FUNCTION_BLOCK MotorVsBase (* Composite Function Block Type *)
  (* Standard: 61499-2 *)
  (* Version 1.0.1, 2/5/2024, ApplicationLibDevTeam, Schneider Electric, First Version *)
  PACKAGE Main;
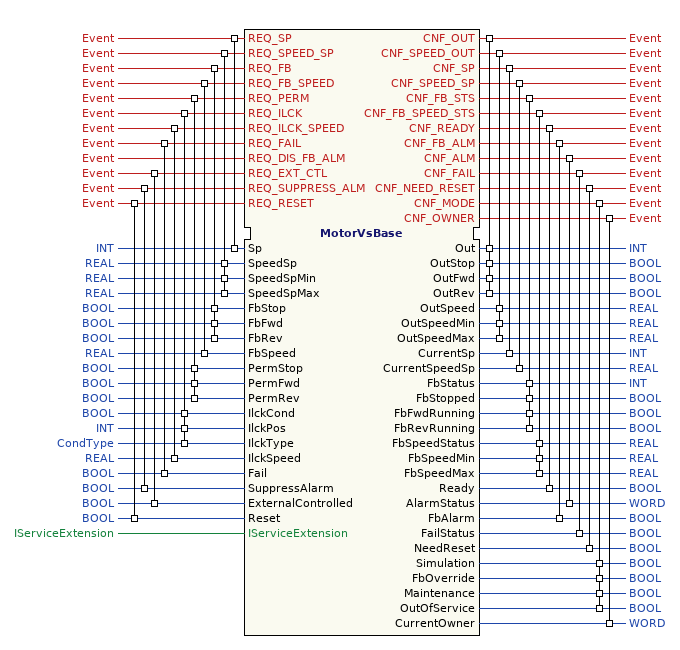
  EVENT_INPUT
    REQ_SP WITH Sp; (* Request to update setpoint *)
    REQ_SPEED_SP WITH SpeedSp, SpeedSpMin, SpeedSpMax;
    REQ_FB WITH FbStop, FbFwd, FbRev; (* Request to update feedbacks *)
    REQ_FB_SPEED WITH FbSpeed;
    REQ_PERM WITH PermStop, PermFwd, PermRev; (* Request to update permissive conditions *)
    REQ_ILCK WITH IlckCond, IlckPos, IlckType; (* Request to update interlock conditions *)
    REQ_ILCK_SPEED WITH IlckSpeed;
    REQ_FAIL WITH Fail; (* Request to update out of service and fail status and parameters *)
    REQ_DIS_FB_ALM; (* Request to disable feedback alarm *)
    REQ_EXT_CTL WITH ExternalControlled; (* Request External control signal *)
    REQ_SUPPRESS_ALM WITH SuppressAlarm; (* Request to update the alarm suppress status *)
    REQ_RESET WITH Reset; (* Request to reset the device *)
  END_EVENT
  EVENT_OUTPUT
    CNF_OUT WITH Out, OutFwd, OutStop, OutRev; (* Execution of output confirmation *)
    CNF_SPEED_OUT WITH OutSpeed, OutSpeedMin, OutSpeedMax; (* Execution of apeed output confirmation *)
    CNF_SP WITH CurrentSp; (* Execution of confirmation current setpoint *)
    CNF_SPEED_SP WITH CurrentSpeedSp; (* Execution of confirmation current speed setpoint *)
    CNF_FB_STS WITH FbFwdRunning, FbStopped, FbStatus, FbRevRunning; (* Execution of confirmed state *)
    CNF_FB_SPEED_STS WITH FbSpeedStatus, FbSpeedMin, FbSpeedMax; (* Execution of confirmed speed state *)
    CNF_READY WITH Ready; (* Execution of ready status *)
    CNF_FB_ALM WITH FbAlarm; (* Execution of confirmation  Fb alarm *)
    CNF_ALM WITH AlarmStatus; (* Execution of confirmation  alarm conditions *)
    CNF_FAIL WITH FailStatus; (* Execution of confirmation  failure *)
    CNF_NEED_RESET WITH NeedReset; (* Request for reset *)
    CNF_MODE WITH Simulation, FbOverride, Maintenance, OutOfService; (* Excecution of new operational modes *)
    CNF_OWNER WITH CurrentOwner; (* Execution confirmation of owner *)
  END_EVENT
  VAR_INPUT
    Sp : INT; (* Setpoint of device (0 = Stop, 1 = Run Forward, 2 = Run Reverse) *)
    SpeedSp : REAL; (* Speed setpoint of device *)
    SpeedSpMin : REAL; (* Speed setpoint minimum range *)
    SpeedSpMax : REAL; (* Speed setpoint maximum range *)
    FbStop : BOOL; (* 1 = Device stop feedback incoming *)
    FbFwd : BOOL; (* 1 = Device forward running feedback incoming *)
    FbRev : BOOL; (* 1 = Device reverse running feedback incoming *)
    FbSpeed : REAL; (* Device speed feedback incoming (Minimum Value  = 0.0, Maximum Value = 100.0) *)
    PermStop : BOOL := TRUE; (* 1 = Device stop permission active *)
    PermFwd : BOOL := TRUE; (* 1 = Device forward run permission active *)
    PermRev : BOOL := TRUE; (* 1 = Device reverse run permission active *)
    IlckCond : BOOL; (* 1 = Interlock condition active *)
    IlckPos : INT; (* Interlock setpoint state (0 = Stop, 1 = Run Forward, 1 = Run Reverse, 3 = Interlock inactive) *)
    IlckType : CondType; (* Type of condition interlock, (0 = Normal, 1 = Process interlock/Sequence interlock) *)
    IlckSpeed : REAL; (* Interlock speed setpoint *)
    Fail : BOOL; (* 1 = Failure is active *)
    SuppressAlarm : BOOL; (* 1 = Suppress alarm in HMI *)
    ExternalControlled : BOOL; (* 1 = External control is active *)
    Reset : BOOL; (* 1 = Reset device failure *)
  END_VAR
  VAR_OUTPUT
    Out : INT; (* Calculated output of the device ( 0 = Stop command, 1 = Forward Run command,  1 = Reverse Run command) *)
    OutStop : BOOL; (* 1 = Stop output of the device *)
    OutFwd : BOOL; (* 1 = Forward output of the device *)
    OutRev : BOOL; (* 1 = Reverse output of the device *)
    OutSpeed : REAL; (* Calculated speed output of the device *)
    OutSpeedMin : REAL; (* Current output speed minimum value *)
    OutSpeedMax : REAL; (* Current output speed maximum value *)
    CurrentSp : INT; (* Current output value considering permissive conditions *)
    CurrentSpeedSp : REAL; (* Current output value *)
    FbStatus : INT; (* Confirmed state of the device (0 = Stopped, 1 =Running, 253 = Unknown) *)
    FbStopped : BOOL; (* 1 = Stopped *)
    FbFwdRunning : BOOL; (* 1 = Running Forward *)
    FbRevRunning : BOOL; (* 1 = Running Reverse *)
    FbSpeedStatus : REAL; (* Speed feedback *)
    FbSpeedMin : REAL; (* Minimum speed setpoint range *)
    FbSpeedMax : REAL; (* Maximum speed setpoint range *)
    Ready : BOOL; (* 1 = Device is ready to run *)
    AlarmStatus : WORD; (* Bit 1 = Device failure status, Bit 2 = Feedback failure status *)
    FbAlarm : BOOL; (* Current output speed minimum value *)
    FailStatus : BOOL; (* 1 = Fail active *)
    NeedReset : BOOL; (* 1 = Device need reset to resume the operation *)
    Simulation : BOOL; (* 1 = Simulation mode is active *)
    FbOverride : BOOL; (* 1 = Feedback overide (Sp = FbStatus) *)
    Maintenance : BOOL; (* 1 = Maintenance mode is active *)
    OutOfService : BOOL; (* 1 = Out of service mode is active *)
    CurrentOwner : WORD; (* Current owner data from externlal source and basic owner 16#8 = Program owner, 16#10 = Operator owner, 16#4 = program Local and 16#40 Operator Local *)
  END_VAR
  SOCKETS
    IServiceExtension : IServiceExtension(ServiceState := TRUE); (* Services extension adapter(Seq control, Local panel, Maintenance and Owner) *)
  END_SOCKETS
  (* Alarm Managment *)
  (* Control *)
  (* Data exchange with sequence *)
  (* Initialization *)
  (* Supervision Interface *)
  (* Owner & Setpoint Management *)
  (* Speed Input *)
  (* Comment If external owner is enabled, the owner for speed selection will be decoupled from normal owner. The external speed owner can be configured from HMI *)
  FBS
    plcStart : plcStart(Delay := T#0ms, Prio := 16);
    IThis : MotorVsBase_HMI(QI := TRUE);
    spSelection : devInSel(EnBumpless2 := TRUE, EnBumpless3 := FALSE); {SET_ATTRIBUTE(Configuration.Component.HideUnusedPorts, )}
    control : motorVsLogic; {SET_ATTRIBUTE(Configuration.Component.HideUnusedPorts, )}
    basicOwner : ownerControl;
    deviceFailure : stateAlarmBasic(AlarmState := TRUE); {SET_ATTRIBUTE(HMI.AlarmText, $key:SE.App2CommonProcess.AlmLableMotorFail)}
    feedbackFailure : stateAlarmBasic(AlarmState := TRUE); {SET_ATTRIBUTE(HMI.AlarmText, $key:SE.App2CommonProcess.AlarmLabelFbFail)}
    programSpSelection : SELECT_24363B89CFDE21263; {SET_ATTRIBUTE(Configuration.GenericFBType.InterfaceParams, Runtime.Standard#CNT:=2;SELECT:BOOL;IN${CNT$}:INT)}
    speedOwner : externalOwnerSel(pin_0E0839046EC8AB65 := TRUE); {SET_ATTRIBUTE(Configuration.Component.HideUnusedPorts, )}
    speedSpSelection : devRealSel(EnBumpless2 := TRUE, EnBumpless3 := FALSE); {SET_ATTRIBUTE(Configuration.Component.HideUnusedPorts, )}
    programSpeedSpSelection : SELECT_218F0E76F8A148ECD; {SET_ATTRIBUTE(Configuration.GenericFBType.InterfaceParams, Runtime.Standard#CNT:=2;SELECT:BOOL;IN${CNT$}:REAL)}
    speedFbScale : limitScaleValue(EnScale := TRUE, UseCutoff := TRUE); {SET_ATTRIBUTE(Configuration.Component.HideUnusedPorts, )}
    speedSpRangeSel : externalRangeSel;
    resetConditions : DS_SELECTX_1579ED5B8ACDFC94C; {SET_ATTRIBUTE(Configuration.GenericFBType.InterfaceParams, Runtime.Standard#CNTX:=3;CNTY:=1;DI${CNTX,_,CNTY$}:BOOL)}
  END_FBS
  EVENT_CONNECTIONS
    spSelection.CNF TO control.REQ_SP;
    control.CNF_OUT TO IServiceExtension.CNF_STATUS;
    control.CNF_FB_STS TO IServiceExtension.CNF_STATUS;
    spSelection.CNF TO IServiceExtension.CNF_STATUS;
    control.CNF_FB_ALM TO CNF_FB_ALM;
    control.CNF_READY TO IServiceExtension.CNF_READY;
    control.CNF_MODE TO IServiceExtension.CNF_OPMODE;
    REQ_SUPPRESS_ALM TO IServiceExtension.CNF_SUPPRESS_ALM;
    REQ_SUPPRESS_ALM TO deviceFailure.REQ_SUPRESS;
    control.CNF_FB_STS TO CNF_FB_STS;
    control.CNF_OUT TO CNF_OUT;
    control.CNF_MODE TO CNF_MODE;
    REQ_FB TO control.REQ_FB;
    REQ_FAIL TO control.REQ_FAIL;
    REQ_DIS_FB_ALM TO control.REQ_PARA;
    deviceFailure.INITO TO feedbackFailure.INIT;
    REQ_PERM TO spSelection.REQ_SEL;
    IServiceExtension.REQ_OWNER TO basicOwner.REQ_STDOWNER;
    basicOwner.CNF_OWNER TO spSelection.REQ_SEL;
    feedbackFailure.INITO TO plcStart.ACK_FIRST;
    control.CNF_NEED_RESET TO CNF_NEED_RESET;
    control.CNF_READY TO CNF_READY;
    spSelection.CNF TO CNF_SP;
    REQ_EXT_CTL TO control.REQ_EXT_CTL;
    control.CNF_FAIL TO deviceFailure.REQ;
    control.CNF_FAIL TO CNF_FAIL;
    plcStart.FIRST_INIT TO IServiceExtension.CNF_SERVICE;
    control.CNF_FB_ALM TO feedbackFailure.REQ;
    control.CNF_ALM TO CNF_ALM;
    control.CNF_ILCK TO spSelection.REQ_SEL;
    control.CNF_FAIL TO spSelection.RESET_SP;
    REQ_SUPPRESS_ALM TO feedbackFailure.REQ_SUPRESS;
    REQ_PERM TO IServiceExtension.CNF_READY;
    basicOwner.CNF_OWNER TO speedOwner.REQ;
    control.CNF_FAIL TO speedSpSelection.RESET_SP;
    REQ_SPEED_SP TO programSpeedSpSelection.REQ;
    IServiceExtension.REQ_SP TO programSpeedSpSelection.REQ;
    control.CNF_ILCK TO speedSpSelection.REQ_SEL;
    speedSpSelection.CNF TO control.REQ_SPEED_SP;
    REQ_ILCK_SPEED TO speedSpSelection.REQ_SEL;
    speedOwner.CNF TO speedSpSelection.REQ_SEL;
    speedFbScale.CNF TO CNF_FB_SPEED_STS;
    IServiceExtension.REQ_OWNER TO speedOwner.REQ;
    REQ_FB_SPEED TO speedFbScale.REQ;
    speedFbScale.CNF TO IServiceExtension.CNF_PV;
    control.CNF_SPEED_OUT TO CNF_SPEED_OUT;
    speedSpSelection.CNF TO CNF_SPEED_SP;
    control.CNF_SPEED_OUT TO IServiceExtension.CNF_SP_OP;
    speedSpSelection.CNF TO IServiceExtension.CNF_SP_OP;
    programSpeedSpSelection.CNF TO speedSpSelection.REQ_SP3;
    REQ_SP TO programSpSelection.REQ;
    IServiceExtension.REQ_CMD TO programSpSelection.REQ;
    programSpSelection.CNF TO spSelection.REQ_SP3;
    control.CNF_ILCK TO IServiceExtension.CNF_READY;
    control.CNF_ALM TO IServiceExtension.CNF_READY;
    control.CNF_NEED_RESET TO IServiceExtension.CNF_READY;
    REQ_ILCK_SPEED TO control.REQ_ILCK_SPEED;
    basicOwner.CNF_OWNER TO speedSpRangeSel.REQ_SELECT;
    speedSpRangeSel.CNF TO control.REQ_SPEED_SP;
    REQ_SPEED_SP TO speedSpRangeSel.REQ_3;
    speedSpRangeSel.CNF TO speedFbScale.REQ;
    IServiceExtension.REQ_SP TO speedSpRangeSel.REQ_2;
    plcStart.FIRST_INIT TO IThis.34A017503AC1070A;
    IThis.377462E9CE5193B5 TO IThis.F2953B6BB9388F21;
    control.CNF_FB_STS TO IThis.EC791CA6E67D66B3;
    control.CNF_OUT TO IThis.EC791CA6E67D66B3;
    control.CNF_NEED_RESET TO IThis.EC791CA6E67D66B3;
    spSelection.CNF TO IThis.EC791CA6E67D66B3;
    control.CNF_TRANS_FB TO IThis.EC791CA6E67D66B3;
    REQ_SUPPRESS_ALM TO IThis.EC791CA6E67D66B3;
    deviceFailure.CNF_ALM TO IThis.EC791CA6E67D66B3;
    feedbackFailure.CNF_ALM TO IThis.EC791CA6E67D66B3;
    control.CNF_FAIL TO IThis.EC791CA6E67D66B3;
    control.CNF_ILCK TO IThis.EC791CA6E67D66B3;
    REQ_PERM TO IThis.EC791CA6E67D66B3;
    basicOwner.CNF_OWNER TO IThis.EC791CA6E67D66B3;
    speedFbScale.CNF TO IThis.EC791CA6E67D66B3;
    control.CNF_SPEED_OUT TO IThis.EC791CA6E67D66B3;
    speedOwner.CNF TO IThis.EC791CA6E67D66B3;
    speedSpSelection.CNF TO IThis.EC791CA6E67D66B3;
    speedSpRangeSel.CNF TO IThis.EC791CA6E67D66B3;
    control.PASSIVE_T TO IThis.FD2B6A321910142C;
    IThis.377462E9CE5193B5 TO deviceFailure.INIT;
    IThis.377462E9CE5193B5 TO basicOwner.REQ_BASICOWNER;
    IThis.B42FC414051FE233 TO basicOwner.REQ_BASICOWNER;
    IThis.1E115F107370F478 TO speedOwner.REQ;
    IThis.1E115F107370F478 TO IServiceExtension.CNF_OWNER;
    IThis.95BEA68906019444 TO control.REQ_PARA;
    IThis.95BEA68906019444 TO feedbackFailure.REQ_PARA;
    IThis.95BEA68906019444 TO deviceFailure.REQ_PARA;
    IThis.95BEA68906019444 TO speedSpRangeSel.REQ_SELECT;
    IThis.A8EC0BB0D1766C60 TO speedSpRangeSel.REQ_1;
    IThis.4BC263E0581D4DDB TO control.REQ_SPEED_SP;
    IThis.C6CA4032A5F6989A TO spSelection.REQ_SP2;
    IThis.369F8CFFBEE23AB4 TO speedSpSelection.REQ_SP2;
    IThis.4711DA9A2DFC024 TO basicOwner.REQ_FORCE;
    IThis.4711DA9A2DFC024 TO control.REQ_PARA;
    IThis.4711DA9A2DFC024 TO spSelection.REQ_SEL;
    IThis.4711DA9A2DFC024 TO speedSpSelection.REQ_SEL;
    REQ_ILCK TO control.REQ_ILCK;
    REQ_EXT_CTL TO IThis.EC791CA6E67D66B3;
    basicOwner.CNF_OWNER TO CNF_OWNER;
    REQ_RESET TO resetConditions.REQ3;
    IServiceExtension.REQ_RESET TO resetConditions.REQ2;
    IThis.1A2B085F4B246BF1 TO resetConditions.REQ1;
    resetConditions.IND TO control.REQ_RESET;
    IThis.95BEA68906019444 TO IServiceExtension.CNF_CFG;
    IThis.A8EC0BB0D1766C60 TO speedFbScale.REQ;
  END_CONNECTIONS
  DATA_CONNECTIONS
    spSelection.PermVal TO control.Sp;
    control.FbStatus TO IServiceExtension.Status;
    spSelection.PermVal TO IServiceExtension.CurrentSp;
    control.Out TO IServiceExtension.CurrentOp;
    control.NeedReset TO IServiceExtension.NeedReset;
    control.FbAlarm TO FbAlarm;
    control.Mode TO IServiceExtension.OpMode;
    control.Ready TO IServiceExtension.Ready;
    SuppressAlarm TO IServiceExtension.SuppressAlarm;
    SuppressAlarm TO deviceFailure.Suppress;
    SuppressAlarm TO feedbackFailure.Suppress;
    control.FbAlarm TO feedbackFailure.Input;
    control.FailStatus TO FailStatus;
    IlckPos TO control.IlckPos;
    IlckType TO control.IlckType;
    FbStop TO control.FbStop;
    FbFwd TO control.FbFwd;
    Fail TO control.Fail;
    PermStop TO spSelection.PermPassive;
    PermFwd TO spSelection.PermActive1;
    control.FbStopped TO FbStopped;
    control.FbFwdRunning TO FbFwdRunning;
    control.Out TO Out;
    control.FbStatus TO FbStatus;
    basicOwner.ProgramOwner TO spSelection.Sel3;
    basicOwner.OperatorOwner TO spSelection.Sel2;
    IlckPos TO spSelection.IlckSp;
    control.Interlocked TO spSelection.Ilck;
    IServiceExtension.StdOwner TO basicOwner.StdOwner;
    basicOwner.StdOwnerConnected TO programSpSelection.SELECT;
    control.NeedReset TO NeedReset;
    control.Ready TO Ready;
    ExternalControlled TO control.ExternalControlled;
    control.FailStatus TO deviceFailure.Input;
    control.AlarmStatus TO AlarmStatus;
    spSelection.PermVal TO CurrentSp;
    control.FailStatus TO spSelection.Fail;
    PermStop TO IServiceExtension.PermPassive;
    PermFwd TO IServiceExtension.PermActive1;
    control.AlarmStatus TO IServiceExtension.Alarm;
    control.Interlocked TO IServiceExtension.Interlocked;
    PermRev TO spSelection.PermActive2;
    basicOwner.Owner TO speedOwner.StdOwner;
    speedOwner.OperOwner TO speedSpSelection.Sel2;
    speedOwner.ProgOwner TO speedSpSelection.Sel3;
    control.Interlocked TO speedSpSelection.Ilck;
    control.FailStatus TO speedSpSelection.Fail;
    basicOwner.StdOwnerConnected TO programSpeedSpSelection.SELECT;
    control.FbRevRunning TO FbRevRunning;
    FbRev TO control.FbRev;
    speedSpSelection.CurrentVal TO control.SpeedSp;
    IlckSpeed TO control.IlckSpeed;
    IlckSpeed TO speedSpSelection.IlckSp;
    speedSpSelection.CurrentVal TO IServiceExtension.CurrentSpReal;
    speedFbScale.PvOut TO FbSpeedStatus;
    control.OutSpeed TO IServiceExtension.CurrentOpReal1;
    speedFbScale.PvOut TO IServiceExtension.Pv;
    IServiceExtension.ExtOwner TO speedOwner.ExtOwner;
    FbSpeed TO speedFbScale.PvIn;
    control.OutSpeedScaled TO OutSpeed;
    speedSpSelection.CurrentVal TO CurrentSpeedSp;
    PermRev TO IServiceExtension.PermActive2;
    SpeedSp TO programSpeedSpSelection.IN1;
    IServiceExtension.SpReal1 TO programSpeedSpSelection.IN2;
    programSpeedSpSelection.OUT TO speedSpSelection.Val3;
    Sp TO programSpSelection.IN1;
    IServiceExtension.Sp TO programSpSelection.IN2;
    programSpSelection.OUT TO spSelection.Val3;
    control.OutFwd TO OutFwd;
    control.OutStop TO OutStop;
    control.OutRev TO OutRev;
    speedSpRangeSel.RangeMin TO control.SpeedSpMin;
    speedSpRangeSel.RangeMin TO speedFbScale.CutoffValue;
    speedSpRangeSel.RangeMin TO speedFbScale.OutMin;
    speedSpRangeSel.RangeMin TO FbSpeedMin;
    speedSpRangeSel.RangeMax TO control.SpeedSpMax;
    speedSpRangeSel.RangeMax TO speedFbScale.OutMax;
    speedSpRangeSel.RangeMax TO FbSpeedMax;
    basicOwner.StdOwnerConnected TO speedSpRangeSel.StdOwnerConnected;
    IServiceExtension.RangeMin TO speedSpRangeSel.RangeMin2;
    IServiceExtension.RangeMax TO speedSpRangeSel.RangeMax2;
    SpeedSpMin TO speedSpRangeSel.RangeMin3;
    SpeedSpMax TO speedSpRangeSel.RangeMax3;
    control.FbStatus TO IThis.E35507CB164A688E;
    control.TransFbStatus TO IThis.937CA40F4D16204B;
    speedFbScale.PvOut TO IThis.5FDD97900C8D5AF7;
    spSelection.PermVal TO IThis.C6876D790F3A950E;
    control.Out TO IThis.D2C35BC47DF71FCC;
    speedSpSelection.CurrentVal TO IThis.977C6234F7727BFD;
    speedSpRangeSel.RangeMin TO IThis.51D483D786BBCC80;
    speedSpRangeSel.RangeMax TO IThis.4209B267B5CDF46;
    control.OutSpeedScaled TO IThis.53DD13BB8E7CA9FB;
    basicOwner.Owner TO IThis.9CB24E1B5B149DBC;
    speedOwner.Owner TO IThis.A2BE276F0EB32372;
    control.NeedReset TO IThis.9CD6749867E91606;
    control.Interlocked TO IThis.22A0744EA4DC0124;
    feedbackFailure.AlarmStatus TO IThis.7F794E74835A9A2;
    deviceFailure.AlarmStatus TO IThis.E4BB2C7DF94BE70A;
    PermStop TO IThis.AB1D2B96094C90BD;
    PermFwd TO IThis.18DA785EF50AD374;
    PermRev TO IThis.49F3F7DCC2A083AE;
    control.PassiveRemainTime TO IThis.1956BBB3F5CBD486;
    basicOwner.StdOwnerConnected TO IThis.621B2EAA60B4DCF6;
    IThis.922C4AB423622B98 TO basicOwner.BasicOwner;
    IThis.4DE40AA7535A5A0C TO speedOwner.EnExtOwner;
    IThis.4DE40AA7535A5A0C TO IServiceExtension.EnExtOwner;
    IThis.7DA82474095F82B2 TO speedOwner.ExtOwnerSel;
    IThis.7DA82474095F82B2 TO IServiceExtension.ExtOwnerSel;
    IThis.861B8773AF2757FC TO control.MonTime;
    IThis.5568E3E91B9AAED8 TO control.TripTime;
    IThis.E0899D0C804160D2 TO control.PassiveTime;
    IThis.3DA6D0F9276D43A4 TO control.ConfResetReq;
    IThis.22AB1FF8E4CF2F97 TO control.FailResetReq;
    IThis.869E02415F6A841 TO spSelection.Val2;
    IThis.5C6A0E86268ED420 TO speedSpSelection.Val2;
    IThis.5508A90160132C15 TO speedSpRangeSel.RangeMin1;
    IThis.2AD891B1627FD8EE TO speedSpRangeSel.RangeMax1;
    IThis.68E0CAABBDF0078 TO control.SpeedOutMin;
    IThis.68E0CAABBDF0078 TO OutSpeedMin;
    IThis.322B60ACD17B29E7 TO control.SpeedOutMax;
    IThis.322B60ACD17B29E7 TO OutSpeedMax;
    IThis.CF1EA84FDDBF53A1 TO control.Simulation;
    IThis.CF1EA84FDDBF53A1 TO Simulation;
    IThis.AD38F01F8F0043E7 TO control.FbOverride;
    IThis.AD38F01F8F0043E7 TO FbOverride;
    IThis.C8DEEF765E4F14C0 TO basicOwner.ForceOperator;
    IThis.C8DEEF765E4F14C0 TO Maintenance;
    IThis.C8DEEF765E4F14C0 TO control.Maintenance;
    IThis.6EDFC17C06F3153 TO spSelection.Sel1;
    IThis.6EDFC17C06F3153 TO OutOfService;
    IThis.6EDFC17C06F3153 TO speedSpSelection.Sel1;
    IThis.6EDFC17C06F3153 TO control.OutOfService;
    IThis.344261B181153C38 TO speedSpRangeSel.Select;
    IThis.152A2BD44E46F288 TO deviceFailure.ScanTime;
    IThis.152A2BD44E46F288 TO feedbackFailure.ScanTime;
    IThis.3CCC10520A21214A TO deviceFailure.AckType;
    IThis.3CCC10520A21214A TO feedbackFailure.AckType;
    IThis.89CD17990DC40B0E TO spSelection.EnTrackSp;
    IThis.89CD17990DC40B0E TO speedSpSelection.EnTrackSp;
    IThis.B2B61A4BABE50F70 TO spSelection.EnResetSp;
    IThis.B2B61A4BABE50F70 TO speedSpSelection.EnResetSp;
    IThis.A07A7C784B98F7E9 TO control.DeviceType;
    IlckCond TO control.IlckCond;
    ExternalControlled TO IThis.C2064A64F1E6B239;
    basicOwner.Owner TO CurrentOwner;
    Reset TO resetConditions.DI3_1;
    IServiceExtension.Reset TO resetConditions.DI2_1;
    IThis.4D34C1A4533BA5DF TO resetConditions.DI1_1;
    resetConditions.OUT1 TO control.Reset;
    IThis.89CD17990DC40B0E TO IServiceExtension.EnTrackSp;
    IThis.B2B61A4BABE50F70 TO IServiceExtension.EnResetSp;
    control.Failure TO IThis.D28866DFD0C1393B;
    IThis.20B18A8DFD1C4D64 TO speedFbScale.InMin;
    IThis.D294948C15C384E1 TO speedFbScale.InMax;
    IThis.5B357E1A1315D6FB TO speedFbScale.4A685434B427A80E;
  END_CONNECTIONS
END_FUNCTION_BLOCK
